{attribute addProperty BoxType "EL3314-0010-0018"}
{attribute addProperty Id "StatusAT %I*Status_F710A6131621ValueAT %I*DINT32417"}
{attribute addProperty CRC "1825988221"}
{attribute addProperty SizeInBites "48"}
{attribute addProperty SizeInBytes "6"}
TYPE TC_Inputs_Channel_6CD65E7D :
STRUCT
	{attribute addProperty Name "Status"}
	Status AT %I* : Status_F710A613;
	{attribute addProperty Name "Value"}
	Value AT %I* : DINT;
END_STRUCT
END_TYPE

(* stored: Version 1.2.0.0, ProductVersion 3.1.4024.9
   DUT TC_Inputs_Channel_6CD65E7D: Id {9be078ee-51d5-4cd1-ac22-a67b107f3905} *)
